Omron CX-Programmer project NewProject (CX-Programmer 9.73)

# PLC NewPLC1: CP1E N20

## Global symbols (name address type ; comment)
0.01 BOOL  ; pb start
0.02 BOOL  ; rs1
0.04 BOOL  ; pb stop
0.05 BOOL  ; rs2
100.00 BOOL  ; cylinder
200.00 BOOL  ; relay
T001 BOOL  ; timer

## Program NewProgram1 (cyclic task 0)

### Section Section1

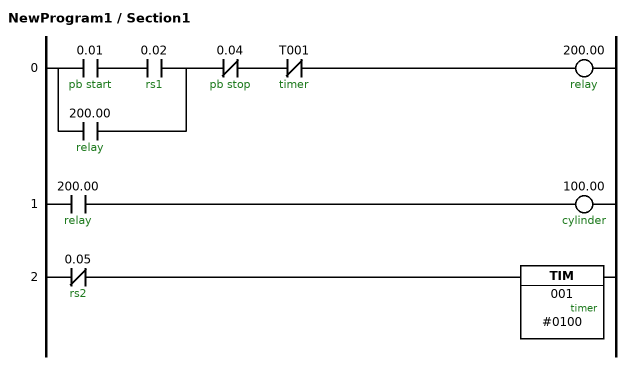
; rung 0
LD 0.01  ; pb start
AND 0.02  ; rs1
OR 200.00  ; relay
ANDNOT 0.04  ; pb stop
ANDNOT T001  ; timer
OUT 200.00  ; relay
; rung 1
LD 200.00  ; relay
OUT 100.00  ; cylinder
; rung 2
LDNOT 0.05  ; rs2
TIM 001 #0100  ; timer

### Section END
; rung 0
END(001)